Staubli VAL3: StackCount.pjx

--- StackCount.pjx ---
Parameters version=s7.9 stackSize=5000 millimeterUnit=true
Program file=recursion.pgx
Program file=recursion1.pgx
Program file=recursion2.pgx
Program file=start.pgx
Program file=stop.pgx
Data file=StackCount.dtx

--- recursion.pgx ---
program recursion()
  local string l_sItem
begin
  nNum=nNum+1
  delay(0.1)
  call recursion()

end
